FUNCTION_BLOCK FB_PTP_AXIS_ABS_CONTROL
VAR_INPUT
	ControlMode:				BOOL;					// Manual (JOG mode) or Automatic (ABSOLUTE PTP mode) | 0:=Manual 1:=Automatic
	
	JogForward:					BOOL;					// Jog the axis in forward direction (based on the JogMode)
	JogBackward:				BOOL;					// Jog the axis in forward direction (based on the JogMode)
	JogMode:					E_JogMode;				// Selected Jog mode is determin the manual movement method stepper or continous
	
	Enable:						BOOL;					// Enable axis
	Start:						BOOL;					// Start to position in automatic mode
	StepSize:					LREAL;					// Stepsize (like: 0.1mm, 0.2mm, 0.5mm, 1mm ....)
	Target:						LREAL;					// Target position in automatic mode
	Override:					LREAL;					// Overall axis override (0-100%)
	ManualOverride:				LREAL;					// Manual override (0-20%)
	MaxVelocity:				LREAL;					// Maximum axis velocity (0-600)
	
	SafetyEnable:				BOOL;
END_VAR
VAR_IN_OUT
	AxisReference:				AXIS_REF;				// Contains all referencies for the NC Axis
END_VAR
VAR_OUTPUT
	Debug:						tsDriveOutputs;			// Debug function block output struct
END_VAR
VAR
	AxisState:					teDriveState;			// Contains the control actual state.
	
	LastTarget:					LREAL;
	
	MoveAbs:					MC_MoveAbsolute;		
	MoveJog:					MC_Jog;
	MoveHalt:					MC_Halt;
	Reset:						MC_Reset;
	SoEReset:					FB_SoEReset;
	Power:						MC_Power;
END_VAR

(* update the axis status at the beginning of each cycle *)
AxisReference();

(* axis drive state machine *)
CASE AxisState OF
	
	MOVESTATE_INIT:																		(* initialisation *)
		MoveAbs.Execute :=			FALSE;
		Reset.Execute :=			FALSE;
		AxisState := 				MOVESTATE_ENABLE;
		
		IF NOT SafetyEnable THEN 
			AxisState := MOVESTATE_ERROR;
		END_IF
	
	MOVESTATE_ENABLE:																	(* enabel power *)
		Power.Enable :=				TRUE;
		Power.BufferMode :=			MC_Aborting;
		
		IF Power.Status THEN
			AxisState := MOVESTATE_IDLE;
		ELSIF Power.Error THEN
			Power.Enable :=				FALSE;
			AxisState := MOVESTATE_ERROR;
		END_IF
	
	MOVESTATE_IDLE:																		(* Idle state stay here until the next command *)			
		IF ControlMode AND Start AND SafetyEnable THEN
			AxisState := MOVESTATE_AUTO;
			
		ELSIF NOT ControlMode AND (JogForward OR JogBackward) AND SafetyEnable THEN
			AxisState := MOVESTATE_MANUAL;
			
		ELSIF NOT SafetyEnable THEN 
			Power.Enable :=				FALSE;
			AxisState := MOVESTATE_ERROR;
		
		END_IF
		
	MOVESTATE_AUTO:																		(* automatic movment mode *)
		IF LastTarget=target AND NOT Start THEN
			AxisState := MOVESTATE_IDLE;
		ELSE
			MoveAbs.Position := 	target;
			MoveAbs.Velocity := 	MaxVelocity;
			MoveAbs.BufferMode := 	MC_Aborting;
			MoveAbs.Execute := 		TRUE;
			
			IF MoveAbs.Done AND NOT Start THEN
				MoveAbs.Execute := FALSE;
				AxisState := MOVESTATE_IDLE;
				
			ELSIF MoveAbs.CommandAborted OR MoveAbs.Error THEN
				AxisState := MOVESTATE_ERROR;
			END_IF	
		END_IF
	
	MOVESTATE_MANUAL:																	(* manual movement mode *)
		MoveJog.Position := 	StepSize;
		MoveJog.Mode := 		JogMode;
		MoveJog.Velocity := 	(ManualOverride*MaxVelocity)/100;						(* speed reduction in manual movement mode *)
		
		IF MoveJog.Done AND NOT MoveHalt.Done THEN
			MoveHalt.Execute := 	TRUE;
			MoveHalt.BufferMode := 	MC_Aborting;
			
		ELSIF MoveHalt.Done AND NOT MoveJog.Done THEN
				MoveHalt.Execute := FALSE;
				AxisState := MOVESTATE_IDLE;

		ELSIF MoveJog.CommandAborted OR MoveAbs.Error OR MoveHalt.CommandAborted THEN
				AxisState := MOVESTATE_ERROR;	
		END_IF
	
	MOVESTATE_ERROR:																	(* in error state *)
		IF AxisReference.Status.Error THEN
			AxisState := MOVESTATE_RESET;												(* axis error requires reset *)
			
		ELSE
			AxisState := MOVESTATE_INIT;												(* function block errors don't need a reset *)
			
		END_IF
	
	MOVESTATE_RESET:																	(* reset axis functions *)
		Power.Enable :=				FALSE;		
		SoEReset.Execute := TRUE;
		SoEReset.Timeout := T#10S;
		IF NOT SoEReset.Busy THEN
			SoEReset.Execute := FALSE;
			Reset.Execute := TRUE;
			IF Reset.Done THEN
				AxisState := MOVESTATE_INIT;	
			ELSIF Reset.Error THEN
				AxisState := MOVESTATE_INIT; 												(* can't do anything here *)
			END_IF
		END_IF
	
END_CASE

ACT_MOVE();
ACT_POWER();
ACT_RESET();

ACTION ACT_MOVE:
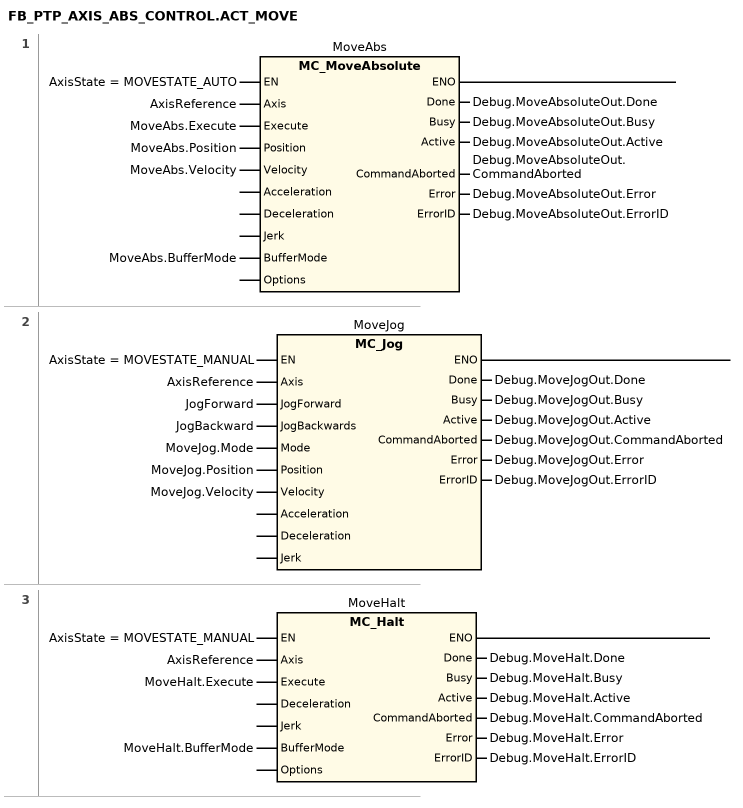
// NETWORK 1
IF AxisState = MOVESTATE_AUTO THEN
    MoveAbs(
        Axis := AxisReference,
        Execute := MoveAbs.Execute,
        Position := MoveAbs.Position,
        Velocity := MoveAbs.Velocity,
        BufferMode := MoveAbs.BufferMode,
        Done => Debug.MoveAbsoluteOut.Done,
        Busy => Debug.MoveAbsoluteOut.Busy,
        Active => Debug.MoveAbsoluteOut.Active,
        CommandAborted => Debug.MoveAbsoluteOut.CommandAborted,
        Error => Debug.MoveAbsoluteOut.Error,
        ErrorID => Debug.MoveAbsoluteOut.ErrorID); // MC_MoveAbsolute
END_IF

// NETWORK 2
IF AxisState = MOVESTATE_MANUAL THEN
    MoveJog(
        Axis := AxisReference,
        JogForward := JogForward,
        JogBackwards := JogBackward,
        Mode := MoveJog.Mode,
        Position := MoveJog.Position,
        Velocity := MoveJog.Velocity,
        Done => Debug.MoveJogOut.Done,
        Busy => Debug.MoveJogOut.Busy,
        Active => Debug.MoveJogOut.Active,
        CommandAborted => Debug.MoveJogOut.CommandAborted,
        Error => Debug.MoveJogOut.Error,
        ErrorID => Debug.MoveJogOut.ErrorID); // MC_Jog
END_IF

// NETWORK 3
IF AxisState = MOVESTATE_MANUAL THEN
    MoveHalt(
        Axis := AxisReference,
        Execute := MoveHalt.Execute,
        BufferMode := MoveHalt.BufferMode,
        Done => Debug.MoveHalt.Done,
        Busy => Debug.MoveHalt.Busy,
        Active => Debug.MoveHalt.Active,
        CommandAborted => Debug.MoveHalt.CommandAborted,
        Error => Debug.MoveHalt.Error,
        ErrorID => Debug.MoveHalt.ErrorID); // MC_Halt
END_IF
END_ACTION

ACTION ACT_POWER:
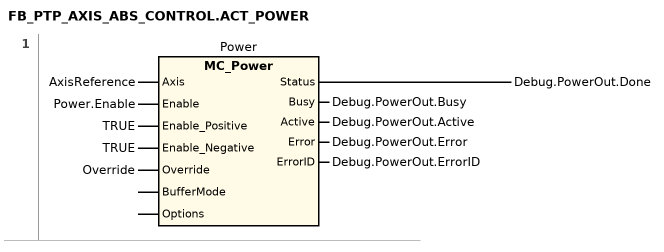
// NETWORK 1
Power(
    Axis := AxisReference,
    Enable := Power.Enable,
    Enable_Positive := TRUE,
    Enable_Negative := TRUE,
    Override := Override,
    Busy => Debug.PowerOut.Busy,
    Active => Debug.PowerOut.Active,
    Error => Debug.PowerOut.Error,
    ErrorID => Debug.PowerOut.ErrorID); // MC_Power
Debug.PowerOut.Done := Power.Status;
END_ACTION

ACTION ACT_RESET:
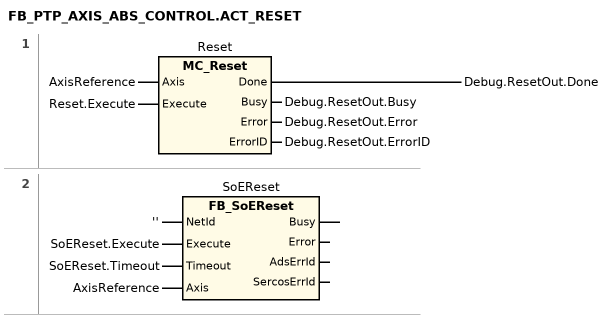
// NETWORK 1
Reset(
    Axis := AxisReference,
    Execute := Reset.Execute,
    Busy => Debug.ResetOut.Busy,
    Error => Debug.ResetOut.Error,
    ErrorID => Debug.ResetOut.ErrorID); // MC_Reset
Debug.ResetOut.Done := Reset.Done;

// NETWORK 2
SoEReset(NetId := '', Execute := SoEReset.Execute, Timeout := SoEReset.Timeout, Axis := AxisReference); // FB_SoEReset
END_ACTION

END_FUNCTION_BLOCK

(* stored: Version 1.1.0.1, ProductVersion 3.1.4022.18
   POU FB_PTP_AXIS_ABS_CONTROL: Id {72ad6629-f379-4e74-8d00-94cd764eedfb}, SpecialFunc None
   Action ACT_MOVE: Id {329169d9-78e7-4a38-829b-c4e8b6fbeb09}
   Action ACT_POWER: Id {2e44ae7d-e511-4e29-b122-f00bb6892c36}
   Action ACT_RESET: Id {9f734f61-7209-405e-a764-135ab4ef3688} *)
